(* IEC 61131-3 sources: Word/plc-course/01-what-is-a-plc/labs/starter, 2 files *)

(* ---- 01-1-lamps-and-switches.st ---- *)
(* Lab 01-1: Lamps and switches - Boolean logic and the lab workflow.
   Module 01 (What is a PLC?). STARTER - the declarations are done for you;
   write the logic where it says TODO, then run:
     python3 tools/plctest.py 01-what-is-a-plc/labs/starter/01-1-lamps-and-switches.st *)

PROGRAM LampsAndSwitches
  VAR (* I/O - addresses follow the OpenPLC convention *)
    SwitchA    AT %IX0.0 : BOOL;  (* Toggle switch A: TRUE when switched on *)
    SwitchB    AT %IX0.1 : BOOL;  (* Toggle switch B: TRUE when switched on *)
    LampTestPB AT %IX0.2 : BOOL;  (* Lamp-test push-button, NO: TRUE while pressed *)
    LampFollow  AT %QX0.0 : BOOL; (* On when switch A is on *)
    LampInverse AT %QX0.1 : BOOL; (* On when switch A is off *)
    LampBoth    AT %QX0.2 : BOOL; (* On when switches A and B are both on *)
    LampEither  AT %QX0.3 : BOOL; (* On when switch A or B (or both) is on *)
  END_VAR

  (* TODO: replace these placeholder lines with one expression per lamp.
     Remember the lamp-test button (requirement 5).
     (MATIEC needs at least one statement in a program body.) *)
  LampFollow  := FALSE;
  LampInverse := FALSE;
  LampBoth    := FALSE;
  LampEither  := FALSE;
END_PROGRAM

CONFIGURATION Config0
  RESOURCE Res0 ON PLC
    TASK MainTask(INTERVAL := T#10ms, PRIORITY := 0);
    PROGRAM Inst0 WITH MainTask : LampsAndSwitches;
  END_RESOURCE
END_CONFIGURATION

(* ---- 01-2-last-write-wins.st ---- *)
(* Lab 01-2: Last write wins - fix a sump pump program that writes its
   outputs in two places.
   Module 01 (What is a PLC?). STARTER - this is the plant's CURRENT program
   and it has a bug. It compiles, but it fails the acceptance test:
     python3 tools/plctest.py 01-what-is-a-plc/labs/starter/01-2-last-write-wins.st
   Copy it to your work folder, find out why, and restructure the logic so
   that it meets every requirement in the lab sheet. Keep the interface
   (names, types and addresses) exactly as it is. *)

PROGRAM SumpPump
  VAR (* I/O - addresses follow the OpenPLC convention *)
    HandSel       AT %IX0.0 : BOOL;  (* HAND-OFF-AUTO selector: TRUE in HAND *)
    AutoSel       AT %IX0.1 : BOOL;  (* HAND-OFF-AUTO selector: TRUE in AUTO *)
    LevelHigh     AT %IX0.2 : BOOL;  (* LSH float switch: TRUE while the level is above it *)
    LevelHH_NC    AT %IX0.3 : BOOL;  (* LSHH switch, NC: TRUE while the level is NOT high-high *)
    OverloadOK_NC AT %IX0.4 : BOOL;  (* Pump overload relay contact, NC: TRUE while healthy *)
    Pump          AT %QX0.0 : BOOL;  (* Pump motor contactor coil *)
    AlarmLamp     AT %QX0.1 : BOOL;  (* Red common alarm lamp *)
  END_VAR

  (* Rung 1 - automatic operation (original program).
     In AUTO the pump runs while the high-level float is up. *)
  Pump := AutoSel AND LevelHigh AND OverloadOK_NC;

  (* Rung 2 - high-high level alarm (original program). *)
  AlarmLamp := NOT LevelHH_NC;

  (* Rung 3 - HAND operation, added during a later modification.
     In HAND the pump runs whenever the overload is healthy. *)
  Pump := HandSel AND OverloadOK_NC;

  (* Rung 4 - pump overload alarm, added during the same modification. *)
  AlarmLamp := NOT OverloadOK_NC;
END_PROGRAM

CONFIGURATION Config0
  RESOURCE Res0 ON PLC
    TASK MainTask(INTERVAL := T#10ms, PRIORITY := 0);
    PROGRAM Inst0 WITH MainTask : SumpPump;
  END_RESOURCE
END_CONFIGURATION
